# EPICS autosave request: iocBoot/generic_motors_ioc/dbSave/FLU_Di_.req
%
% BURT Request File
%
% $(P)FLU:Di:  Fluorescent Detector Distance
%

file assy.req ASSY=$(P)FLU:Di
file mtr1.req MTR1=$(P)FLU:md
file drv1.req DRV1=$(P)FLU:D
